// TIA Portal V19 export
TYPE "LEXCHANGETRAY_typeHandlingXyzEm_toConstraintRollerFeedback"
// stored: Access Published
   STRUCT
      xPosDone : Bool;   // X轴到位
      catchOut : Bool;   // 电池取走
   END_STRUCT;
END_TYPE
